# EPICS substitutions: NucInstDigApp/Db/NucInstDigTOFSpec.substitutions
global { "P=\$(P)", "Q=\$(Q)" }

file "NucInstDigTOFSpec.template" {
    pattern { N }
    { "1" }
    { "2" }
    { "3" }
    { "4" }
}
